{attribute 'qualified_only'}
VAR_GLOBAL
// FB DRIVE MccRev_019
	bAutoButton  	   : BOOL;  // SCADA button Auto/manual Command
	bForwardButton     : BOOL;  // SCADA button Forward drive Command
	bReverseButton	   : BOOL;  // SCADA button Reverse drive Command	 
	bTermFuse          : BOOL;  // Term Fuse state from psyhical input
	bContactor         : BOOL;  // Contactor state from psyhical output
	udHours   		   : UDINT; // Work Time Counter - hours nonvolatile memory register
	uMinutes	   	   : UINT;  // Work Time Counter - minutes nonvolatile memory registerr
	uSeconds           : UINT;  // Work Time Counter - seconds nonvolatile memory register
  	sStatus	           : T_MaxString; // Motor Status string
	sState 	           : T_MaxString; // Motor State string	

END_VAR

(* stored: Version 1.1.0.1, ProductVersion 3.1.4024.12
   GVL MccRev_018: Id {5e52bb14-c353-4baa-9e78-25218f1b8b15} *)
